{attribute 'OPC.UA.DA.StructuredType' := '1'}
TYPE ST_eChillerState :
STRUCT
	bError : BOOL;
	bWarning: BOOL;
	//implementation is missing, must be added after startup
END_STRUCT
END_TYPE

(* stored: Version 1.1.0.1, ProductVersion 3.1.4024.9
   DUT ST_eChillerState: Id {8fe2498f-481f-455a-a37c-622be90ae6f7} *)
